// Mitsubishi GX Works2 project: n05   PLC: Q02/Q02H

PROGRAM MAIN
VAR
  CTU_1 : CTU;
  CTU_2 : CTU;
END_VAR
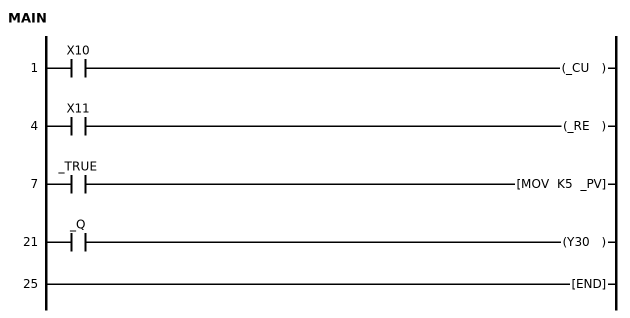
; FB BLK START CTU(CTU_2)
1     LD      X10
      OUT     _CU
4     LD      X11
      OUT     _RE
7     LD      _TRUE
      MOV     K5 _PV
; FB START
; FB_NAME CTU
; INSTANCE_NAME CTU_2
; FB IN_B:CU
; FB OUT_Q:B
; FB IN_B:RE
; FB OUT_CV:W
; FB IN_W:PV
; FB END
21    LD      _Q
      OUT     Y30
; FB BLK END
25    END
END_PROGRAM

FUNCTION_BLOCK CTU
VAR_INPUT
  CU : BOOL;
  RE : BOOL;
  PV : INT;
END_VAR
VAR_OUTPUT
  Q : BOOL;
  CV : INT;
END_VAR
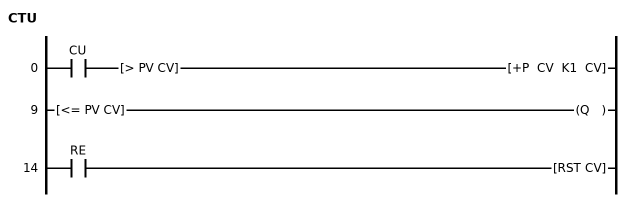
0     LD      CU
      AND>    PV CV
      +P      CV K1 CV
9     LD<=    PV CV
      OUT     Q
14    LD      RE
      RST     CV
END_FUNCTION_BLOCK
